# EPICS substitutions: apps/svtApp/Db/V450-160subnet.substitutions
file "db/HFCBVME-160.db" {
 pattern { N, S, T, H, A, LVD }
  { "0","2","_TEMP","R1S1T_Slot","0","R1S1T_Slot1" }
  { "0","2","_TEMP","R1S1B_Slot","1","R1S1B_Slot1" }
  { "0","2","_TEMP","R1S2T_Slot","2","R1S2T_Slot1" }
  { "0","2","_TEMP","R1S2B_Slot","3","R1S2B_Slot1" }
  { "0","2","_TEMP","R1S3T_Slot","4","R1S3T_Slot2" }
  { "0","2","_TEMP","R1S3B_Slot","5","R1S3B_Slot2" }
  { "0","2","_TEMP","R1S4T_Slot","6","R1S4T_Slot2" }
  { "0","2","_TEMP","R1S4B_Slot","7","R1S4B_Slot2" }
  { "0","2","_TEMP","R1S5T_Slot","8","R1S5T_Slot3" }
  { "0","2","_TEMP","R1S5B_Slot","9","R1S5B_Slot3" }
  { "0","2","_TEMP","R1S6T_Slot","10","R1S6T_Slot3" }
  { "0","2","_TEMP","R1S6B_Slot","11","R1S6B_Slot3" }
  { "0","2","_TEMP","R1S7T_Slot","12","R1S7T_Slot4" }
  { "0","2","_TEMP","R1S7B_Slot","13","R1S7B_Slot4" }
  { "0","2","_TEMP","R1S8T_Slot","14","R1S8T_Slot4" }
  { "0","2","_TEMP","R1S8B_Slot","15","R1S8B_Slot4" }
  { "1","3","_TEMP","R1S9T_Slot","0","R1S9T_Slot5" }
  { "1","3","_TEMP","R1S9B_Slot","1","R1S9B_Slot5" }
  { "1","3","_TEMP","R1S10T_Slot","2","R1S10T_Slot5" }
  { "1","3","_TEMP","R1S10B_Slot","3","R1S10B_Slot5" }
  { "1","3","_TEMP","R2S1T_Slot","4","R2S1T_Slot1" }
  { "1","3","_TEMP","R2S1B_Slot","5","R2S1B_Slot1" }
  { "1","3","_TEMP","R2S2T_Slot","6","R2S2T_Slot1" }
  { "1","3","_TEMP","R2S2B_Slot","7","R2S2B_Slot1" }
  { "1","3","_TEMP","R2S3T_Slot","8","R2S3T_Slot2" }
  { "1","3","_TEMP","R2S3B_Slot","9","R2S3B_Slot2" }
  { "1","3","_TEMP","R2S4T_Slot","10","R2S4T_Slot2" }
  { "1","3","_TEMP","R2S4B_Slot","11","R2S4B_Slot2" }
  { "1","3","_TEMP","R2S5T_Slot","12","R2S5T_Slot3" }
  { "1","3","_TEMP","R2S5B_Slot","13","R2S5B_Slot3" }
  { "1","3","_TEMP","R2S6T_Slot","14","R2S6T_Slot3" }
  { "1","3","_TEMP","R2S6B_Slot","15","R2S6B_Slot3" }
  { "2","4","_TEMP","R2S7T_Slot","0","R2S7T_Slot4" }
  { "2","4","_TEMP","R2S7B_Slot","1","R2S7B_Slot4" }
  { "2","4","_TEMP","R2S8T_Slot","2","R2S8T_Slot4" }
  { "2","4","_TEMP","R2S8B_Slot","3","R2S8B_Slot4" }
  { "2","4","_TEMP","R2S9T_Slot","4","R2S9T_Slot5" }
  { "2","4","_TEMP","R2S9B_Slot","5","R2S9B_Slot5" }
  { "2","4","_TEMP","R2S10T_Slot","6","R2S10T_Slot5" }
  { "2","4","_TEMP","R2S10B_Slot","7","R2S10B_Slot5" }
  { "2","4","_TEMP","R2S11T_Slot","8","R2S11T_Slot6" }
  { "2","4","_TEMP","R2S11B_Slot","9","R2S11B_Slot6" }
  { "2","4","_TEMP","R2S12T_Slot","10","R2S12T_Slot6" }
  { "2","4","_TEMP","R2S12B_Slot","11","R2S12B_Slot6" }
  { "2","4","_TEMP","R2S13T_Slot","12","R2S13T_Slot7" }
  { "2","4","_TEMP","R2S13B_Slot","13","R2S13B_Slot7" }
  { "2","4","_TEMP","R2S14T_Slot","14","R2S14T_Slot7" }
  { "2","4","_TEMP","R2S14B_Slot","15","R2S14B_Slot7" }
  { "3","5","_TEMP","R3S1T_Slot","0","R3S1T_Slot1" }
  { "3","5","_TEMP","R3S1B_Slot","1","R3S1B_Slot1" }
  { "3","5","_TEMP","R3S2T_Slot","2","R3S2T_Slot1" }
  { "3","5","_TEMP","R3S2B_Slot","3","R3S2B_Slot1" }
  { "3","5","_TEMP","R3S3T_Slot","4","R3S3T_Slot2" }
  { "3","5","_TEMP","R3S3B_Slot","5","R3S3B_Slot2" }
  { "3","5","_TEMP","R3S4T_Slot","6","R3S4T_Slot2" }
  { "3","5","_TEMP","R3S4B_Slot","7","R3S4B_Slot2" }
  { "3","5","_TEMP","R3S5T_Slot","8","R3S5T_Slot3" }
  { "3","5","_TEMP","R3S5B_Slot","9","R3S5B_Slot3" }
  { "3","5","_TEMP","R3S6T_Slot","10","R3S6T_Slot3" }
  { "3","5","_TEMP","R3S6B_Slot","11","R3S6B_Slot3" }
  { "3","5","_TEMP","R3S7T_Slot","12","R3S7T_Slot4" }
  { "3","5","_TEMP","R3S7B_Slot","13","R3S7B_Slot4" }
  { "3","5","_TEMP","R3S8T_Slot","14","R3S8T_Slot4" }
  { "3","5","_TEMP","R3S8B_Slot","15","R3S8B_Slot4" }
  { "4","6","_TEMP","R3S9T_Slot","0","R3S9T_Slot5" }
  { "4","6","_TEMP","R3S9B_Slot","1","R3S9B_Slot5" }
  { "4","6","_TEMP","R3S10T_Slot","2","R3S10T_Slot5" }
  { "4","6","_TEMP","R3S10B_Slot","3","R3S10B_Slot5" }
  { "4","6","_TEMP","R3S11T_Slot","4","R3S11T_Slot6" }
  { "4","6","_TEMP","R3S11B_Slot","5","R3S11B_Slot6" }
  { "4","6","_TEMP","R3S12T_Slot","6","R3S12T_Slot6" }
  { "4","6","_TEMP","R3S12B_Slot","7","R3S12B_Slot6" }
  { "4","6","_TEMP","R3S13T_Slot","8","R3S13T_Slot7" }
  { "4","6","_TEMP","R3S13B_Slot","9","R3S13B_Slot7" }
  { "4","6","_TEMP","R3S14T_Slot","10","R3S14T_Slot7" }
  { "4","6","_TEMP","R3S14B_Slot","11","R3S14B_Slot7" }
  { "4","6","_TEMP","R3S15T_Slot","12","R3S15T_Slot8" }
  { "4","6","_TEMP","R3S15B_Slot","13","R3S15B_Slot8" }
  { "4","6","_TEMP","R3S16T_Slot","14","R3S16T_Slot8" }
  { "4","6","_TEMP","R3S16B_Slot","15","R3S16B_Slot8" }
  { "5","7","_TEMP","R3S17T_Slot","0","R3S17T_Slot9" }
  { "5","7","_TEMP","R3S17B_Slot","1","R3S17B_Slot9" }
  { "5","7","_TEMP","R3S18T_Slot","2","R3S18T_Slot9" }
  { "5","7","_TEMP","R3S18B_Slot","3","R3S18B_Slot9" }
  { "6","8","_TEMP","R4S1T_Slot","0","R4S1T_Slot1" }
  { "6","8","_TEMP","R4S1B_Slot","1","R4S1B_Slot1" }
  { "6","8","_TEMP","R4S2T_Slot","2","R4S2T_Slot1" }
  { "6","8","_TEMP","R4S2B_Slot","3","R4S2B_Slot1" }
  { "6","8","_TEMP","R4S3T_Slot","4","R4S3T_Slot2" }
  { "6","8","_TEMP","R4S3B_Slot","5","R4S3B_Slot2" }
  { "6","8","_TEMP","R4S4T_Slot","6","R4S4T_Slot2" }
  { "6","8","_TEMP","R4S4B_Slot","7","R4S4B_Slot2" }
  { "6","8","_TEMP","R4S5T_Slot","8","R4S5T_Slot3" }
  { "6","8","_TEMP","R4S5B_Slot","9","R4S5B_Slot3" }
  { "6","8","_TEMP","R4S6T_Slot","10","R4S6T_Slot3" }
  { "6","8","_TEMP","R4S6B_Slot","11","R4S6B_Slot3" }
  { "6","8","_TEMP","R4S7T_Slot","12","R4S7T_Slot4" }
  { "6","8","_TEMP","R4S7B_Slot","13","R4S7B_Slot4" }
  { "6","8","_TEMP","R4S8T_Slot","14","R4S8T_Slot4" }
  { "6","8","_TEMP","R4S8B_Slot","15","R4S8B_Slot4" }
  { "7","9","_TEMP","R4S9T_Slot","0","R4S9T_Slot5" }
  { "7","9","_TEMP","R4S9B_Slot","1","R4S9B_Slot5" }
  { "7","9","_TEMP","R4S10T_Slot","2","R4S10T_Slot5" }
  { "7","9","_TEMP","R4S10B_Slot","3","R4S10B_Slot5" }
  { "7","9","_TEMP","R4S11T_Slot","4","R4S11T_Slot6" }
  { "7","9","_TEMP","R4S11B_Slot","5","R4S11B_Slot6" }
  { "7","9","_TEMP","R4S12T_Slot","6","R4S12T_Slot6" }
  { "7","9","_TEMP","R4S12B_Slot","7","R4S12B_Slot6" }
  { "7","9","_TEMP","R4S13T_Slot","8","R4S13T_Slot1" }
  { "7","9","_TEMP","R4S13B_Slot","9","R4S13B_Slot1" }
  { "7","9","_TEMP","R4S14T_Slot","10","R4S14T_Slot1" }
  { "7","9","_TEMP","R4S14B_Slot","11","R4S14B_Slot1" }
  { "7","9","_TEMP","R4S15T_Slot","12","R4S15T_Slot2" }
  { "7","9","_TEMP","R4S15B_Slot","13","R4S15B_Slot2" }
  { "7","9","_TEMP","R4S16T_Slot","14","R4S16T_Slot2" }
  { "7","9","_TEMP","R4S16B_Slot","15","R4S16B_Slot2" }
  { "8","10","_TEMP","R4S17T_Slot","0","R4S17T_Slot3" }
  { "8","10","_TEMP","R4S17B_Slot","1","R4S17B_Slot3" }
  { "8","10","_TEMP","R4S18T_Slot","2","R4S18T_Slot3" }
  { "8","10","_TEMP","R4S18B_Slot","3","R4S18B_Slot3" }
  { "8","10","_TEMP","R4S19T_Slot","4","R4S19T_Slot4" }
  { "8","10","_TEMP","R4S19B_Slot","5","R4S19B_Slot4" }
  { "8","10","_TEMP","R4S20T_Slot","6","R4S20T_Slot4" }
  { "8","10","_TEMP","R4S20B_Slot","7","R4S20B_Slot4" }
  { "8","10","_TEMP","R4S21T_Slot","8","R4S21T_Slot5" }
  { "8","10","_TEMP","R4S21B_Slot","9","R4S21B_Slot5" }
  { "8","10","_TEMP","R4S22T_Slot","10","R4S22T_Slot5" }
  { "8","10","_TEMP","R4S22B_Slot","11","R4S22B_Slot5" }
  { "8","10","_TEMP","R4S23T_Slot","12","R4S23T_Slot6" }
  { "8","10","_TEMP","R4S23B_Slot","13","R4S23B_Slot6" }
  { "8","10","_TEMP","R4S24T_Slot","14","R4S24T_Slot6" }
  { "8","10","_TEMP","R4S24B_Slot","15","R4S24B_Slot6" }
 }
